// This function has been automatically generated from the project information.
{attribute 'signature_flag' := '1073741824'}
{attribute 'TcGenerated'}
{attribute 'no-analysis'}
FUNCTION F_GetVersion : ST_LibVersion
VAR_INPUT
	
END_VAR

F_GetVersion.iMajor := 16;
F_GetVersion.iMinor := 0;
F_GetVersion.iBuild := 2;
F_GetVersion.iRevision := 0;
F_GetVersion.sVersion := '16.0.2';
F_GetVersion.nFlags := 1;

END_FUNCTION

(* stored: Version 1.1.0.1
   POU F_GetVersion: Id {703614b3-d2b1-47c6-b69a-498531a442a4}, SpecialFunc None *)
